FUNCTION_BLOCK FB_Medir_SFC

VAR_INPUT
    // SFC-Flags
    SFCPause: BOOL;
    SFCReset: BOOL;

    // Sincronizacion
    Benido: BOOL ;
    Ejecuta: BOOL;
    DetectorFotoelectrico AT %I*:BOOL;
     DetectorInductivo AT %I*:BOOL;
	MedidorAltura AT %I* : UINT;
   END_VAR
VAR_OUTPUT
	
	// Sincronizacion    
    Acabhe: BOOL;
    ListoKalisto: BOOL;
	MedidorBaja: BOOL;
    END_VAR
VAR_IN_OUT
    // Tapas: (METALICAS, BLANCAS, NEGRAS, ALTAS, BAJAS);
    Tapas : ARRAY[0..7] OF ST_POSICION;
END_VAR

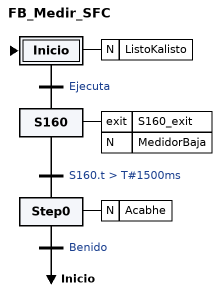
INITIAL_STEP Inicio:
    ListoKalisto(N);
END_STEP
TRANSITION FROM Inicio TO S160
    := Ejecuta;
END_TRANSITION
STEP S160:
    S160_exit(P0);  // exit action
    MedidorBaja(N);
END_STEP
TRANSITION FROM S160 TO Step0
    := S160.t > T#1500ms;
END_TRANSITION
STEP Step0:
    Acabhe(N);
END_STEP
TRANSITION FROM Step0 TO Inicio
    := Benido;
END_TRANSITION

ACTION S160_exit:
Tapas[2].Tapa.Alta := (MedidorAltura <= 1300);
Tapas[3].Tapa.Clara := DetectorFotoelectrico;
Tapas[4].Tapa.Metalica := DetectorInductivo;
END_ACTION

END_FUNCTION_BLOCK

(* stored: Version 1.1.0.1, ProductVersion 3.1.4024.12
   POU FB_Medir_SFC: Id {f90a7250-1615-43c4-95f4-0e149e6a705b}, SpecialFunc None
   Action S160_exit: Id {90d42629-8dd0-43db-830d-c27c6edab4ce} *)
